FUNCTION_BLOCK FB_MasterRobot
VAR_INPUT
END_VAR
VAR_OUTPUT
END_VAR
VAR
	// arm shoulders frame in monitor
	m_shoulderPose :ARRAY[1..2] OF ST_Frame;
	
	// master arms, responsible for arm kinematic and control
	m_masterArms :ARRAY[1..2] OF FB_MasterArm;
	
	// current and las arm state
	m_masterArmState:ARRAY[1..2] OF E_masterArmState:=[E_masterArmState.MasterArmState_Init,E_masterArmState.MasterArmState_Init];
	m_lastMasterArmState:ARRAY[1..2] OF E_masterArmState:=[E_masterArmState.MasterArmState_Init,E_masterArmState.MasterArmState_Init];
	
	// index(1 to 4) of slave arm which is tele-linked to master arm
	m_slaveArmIdx:ARRAY[1..2] OF E_MatchedSlaveArmIdx:=[MatchedSlaveArmIdx_NULL, MatchedSlaveArmIdx_null];
	
	// arm controller
	m_armCtrl :I_MasterArmCtrl;
END_VAR

METHOD PUBLIC Init : BOOL
VAR_INPUT
END_VAR
VAR
	i:INT;
END_VAR
FOR i:=1 TO g_mArmNum DO
	m_masterArms[i].Init(i);
	m_masterArmState[i]:=MasterArmState_Init;
	m_lastMasterArmState[i]:=MasterArmState_Init;
	m_slaveArmIdx[i]:=MatchedSlaveArmIdx_NULL;
END_FOR

m_shoulderPose[1].m_pos[1]:= g_armShoulderDistance/2.0;
m_shoulderPose[2].m_pos[1]:= -g_armShoulderDistance/2.0;
END_METHOD

METHOD PUBLIC run : BOOL
VAR_IN_OUT CONSTANT
	i_cartStatus :ST_CartStatus;
	
	i_slaveStatus :ST_SlaveStatus;
END_VAR
VAR
	i:INT;
END_VAR
// state machine transition
stateMachine(i_cartStatus,i_slaveStatus);

// update shoulder pose (wrt monitor)
m_shoulderPose[1].m_rot:=rotY(m_shoulderPose[1].m_rot,i_cartStatus.m_monitorAngle);
m_shoulderPose[2].m_rot:=rotY(m_shoulderPose[2].m_rot,i_cartStatus.m_monitorAngle);

// update master arm kinematics
FOR i:=1 TO g_mArmNum DO
	m_masterArms[i].updateStatus();
END_FOR

// run controller
m_armCtrl.run(m_shoulderPose,i_slaveStatus, m_masterArms);

// update commands to drivers
FOR i:=1 TO g_mArmNum DO
	m_masterArms[i].updateCmds();
END_FOR
END_METHOD

// state machine check and transit 
METHOD PROTECTED stateMachine : BOOL
VAR_IN_OUT CONSTANT
	i_cartStatus :ST_CartStatus;
	
	i_slaveStatus :ST_SlaveStatus;
END_VAR
END_METHOD

END_FUNCTION_BLOCK

(* stored: Version 1.1.0.1, ProductVersion 3.1.4024.12
   POU FB_MasterRobot: Id {8cbdb2ba-9735-46e3-8cbc-296330acc8cc}, SpecialFunc None
   Method Init: Id {610a17f3-34c5-4e3c-bbbc-19f9c2f46946}
   Method run: Id {ed6f787a-4dc0-4602-b386-92a3c3880a23}
   Method stateMachine: Id {b9cc8560-9309-49e3-93b5-28cb02b4f5cc} *)
